FUNCTION_BLOCK FB_MotionErrorCodeLookup_Test EXTENDS TcUnit.FB_TestSuite
VAR
    Expected: BOOL := True;
    Actual: BOOL;
END_VAR

TEST('FB_MotionErrorCodeLookup_Test Dummy Test');
AssertEquals(Expected := Expected,
             Actual := Actual,
             Message := 'Error Message');
TEST_FINISHED();

END_FUNCTION_BLOCK

(* stored: Version 1.1.0.1, ProductVersion 3.1.4022.18
   POU FB_MotionErrorCodeLookup_Test: Id {c2d62f22-4956-4b9a-a49c-f0bce1724eed}, SpecialFunc None *)
